(* PLC project PLC, Beckhoff Automation GmbH TwinCAT PLC Control 3.5.20.60 *)
(* stored: creationDateTime 2026-07-21T08:44:21.1643744, modificationDateTime 2026-07-21T08:44:21.1643744 *)

TYPE ST_ADS_API_ScadaViewerApp_PLC_In :

STRUCT

	Status				:	ST_ADS_API_ScadaViewerApp_PLC_In_Status;	// |1| Status PC aplikace
	
END_STRUCT

END_TYPE
